TYPE ST_Safety :
STRUCT
    stSafetyIn: ST_SafetyIn;
    stSafetyOut: ST_SafetyOut;
END_STRUCT
END_TYPE

(* stored: Version 1.1.0.1
   DUT ST_Safety: Id {a14bb73e-e071-0777-120d-26666a0ac858} *)
